(* IEC 61131-3 sources: OpenPlc_Lezioni/, 10 files *)

(* ---- Conter.st ---- *)
TYPE
  LOGLEVEL : (CRITICAL, WARNING, INFO, DEBUG) := INFO;
END_TYPE

FUNCTION_BLOCK LOGGER
  VAR_INPUT
    TRIG : BOOL;
    MSG : STRING;
    LEVEL : LOGLEVEL := INFO;
  END_VAR
  VAR
    TRIG0 : BOOL;
  END_VAR

  IF TRIG AND NOT TRIG0 THEN
  {{
   LogMessage(GetFbVar(LEVEL),(char*)GetFbVar(MSG, .body),GetFbVar(MSG, .len));
  }}
  END_IF;
  TRIG0:=TRIG;
END_FUNCTION_BLOCK

PROGRAM program0
  VAR
    CTU0 : CTU;
  END_VAR
  VAR
    BT1 : BOOL;
    BT2 : BOOL;
    Led : BOOL;
  END_VAR
  VAR
    PV : INT := 5;
    R_TRIG1 : R_TRIG;
  END_VAR

  R_TRIG1(CLK := BT1);
  CTU0(CU := R_TRIG1.Q, R := BT2, PV := PV);
  Led := CTU0.Q;
END_PROGRAM

CONFIGURATION Config0

  RESOURCE Res0 ON PLC
    TASK task0(INTERVAL := T#20ms,PRIORITY := 0);
    PROGRAM instance0 WITH task0 : program0;
  END_RESOURCE
END_CONFIGURATION

(* ---- Conunt.st ---- *)
VAR
    AVANTI : BOOL;
    INDIETRO : BOOL;
    RESET : BOOL;
    CONT1 : CTUD;
END_VAR

CONT1(
    CU := AVANTI,
    CD := INDIETRO,
    RESET := RESET,
    LOAD := FALSE,
    PV := 10
);

(* ---- Conut_UP.st ---- *)
VAR
    AVANTI : BOOL;
    INDIETRO : BOOL;
    MIO_RESET: BOOL;
    CONT1 : CTUD;
    VALORE_ATTUALE : INT;
    LIMITE_RAGGIUNTO : BOOL;
END_VAR

// Chiamata del blocco contatore Up/Down
CONT1(
    CU := AVANTI,
    CD := INDIETRO,
    R := MIO_RESET,
    LD := FALSE,
    PV := 10
);

// Lettura delle uscite del blocco
VALORE_ATTUALE := CONT1.CV; // Valore attuale del conteggio
LIMITE_RAGGIUNTO := CONT1.QU; // True se CV >= PV (10)

(* ---- Count_indietro.st ---- *)
VAR
    INDIETRO : BOOL;
    RESET : BOOL;
    CONT1 : CTUD;
END_VAR

CONT1(
    CU := FALSE,
    CD := INDIETRO,
    RESET := RESET,
    LOAD := FALSE,
    PV := 10
);

(* ---- Count_led.st ---- *)
VAR
    AVANTI : BOOL;
    INDIETRO : BOOL;
    RESET : BOOL;
    CONTATORE : INT;
    LED : BOOL;
END_VAR

IF RESET THEN
    CONTATORE := 0;
ELSE
    IF AVANTI THEN
        CONTATORE := CONTATORE + 1;
    ELSE
        IF INDIETRO THEN
            IF CONTATORE > 0 THEN
                CONTATORE := CONTATORE - 1;
            END_IF;
        END_IF;
    END_IF;
END_IF;

// LED acceso quando il contatore arriva a 10
LED := CONTATORE >= 10;

(* ---- Tof2.st ---- *)
VAR
    S1 : BOOL;
    LED : BOOL;
    TOF1 : TOF;
END_VAR

TOF1(IN := S1, PT := T#5s);

IF TOF1.Q THEN
    LED := TRUE;
ELSE
    LED := FALSE;
END_IF;

(* ---- Tof_Plc.st ---- *)
VAR
S1 : BOOL;
LED : BOOL;
TOF1 : TOF;
END_VAR

TOF1(IN := S1, PT := T#5s);

LED := TOF1.Q;

(* ---- TonLed.st ---- *)
VAR
    S1 : BOOL; // Pulsante
    LED1 : BOOL; // LED
    TON1 : TON; // Timer TON
END_VAR

// Avvio temporizzatore quando premo S1
TON1(IN := S1, PT := T#5s);

// Accendo il LED quando il timer è terminato
LED1 := TON1.Q;

(* ---- TONR.st ---- *)
VAR
    S1 : BOOL;
    RESET : BOOL;
    LED : BOOL;
    TONR1 : TONR;
END_VAR

TONR1(IN := S1, R := RESET, PT := T#10s);

IF TONR1.Q THEN
    LED := TRUE;
ELSE
    LED := FALSE;
END_IF;

(* ---- Tp_ftimer.st ---- *)
VAR
    S1 : BOOL;
    LED : BOOL;
    TP1 : TP;
END_VAR

TP1(IN := S1, PT := T#5s);

IF TP1.Q THEN
    LED := TRUE;
ELSE
    LED := FALSE;
END_IF;
